// TIA Portal V17 export
// export: Created 2025-06-20T10:18:27.2090798Z, ExportSetting WithDefaults, DisplayName Totally Integrated Automation Portal, DisplayVersion V17 Update 8, DisplayName TIA Portal Openness, DisplayVersion V17 Update 8, DisplayName TIA Portal Version Control Interface, DisplayVersion V17, DisplayName SINAMICS Startdrive Advanced, DisplayVersion V17 SP2, DisplayName SINAMICS Startdrive G110M, G120, G120C, G120D, G120P, G115D, DisplayVersion V17 SP2, DisplayName SINAMICS Startdrive G130, G150, S120, S150, SINAMICS MV, S210, DisplayVersion V17 SP2, DisplayName STEP 7 Professional, DisplayVersion V17 Update 8, DisplayName SINUMERIK ONE STEP 7 Toolbox, DisplayVersion V17 Update 12, DisplayName SINUMERIK ONE PLC Basic Program Plus, DisplayVersion V17 Update 12, DisplayName SINUMERIK 840D sl STEP 7 Toolbox, DisplayVersion V17 Update 12, DisplayName STEP 7 Safety, DisplayVersion V17 Update 6, DisplayName WinCC Advanced, DisplayVersion V17 Update 8
DATA_BLOCK "DB17100_MAINTENANCE_OPERATOR_HELP"   // DB17100
{ S7_Optimized_Access := 'TRUE'; DB_Accessible_From_OPC_UA := 'FALSE' }
VERSION : 0.1
// stored: AutoNumber false, DBAccessibleFromOPCUA false, DBAccessibleFromWebserver true, IsOnlyStoredInLoadMemory false, IsRetainMemResEnabled false, IsWriteProtectedInAS false, MemoryReserve 100
   VAR
      OPERATOR_HELP : Array[0..100] of Bool;
   END_VAR
BEGIN
   // OPERATOR_HELP[0] : MAINTENANCE OPERATOR HELP
   // OPERATOR_HELP[1] : POWDER > UNIT 1 > GENERAL -- UNIT 1 ACTION IN TUBE OF SECTION 4
   // OPERATOR_HELP[2] : POWDER > UNIT 1 > GENERAL -- UNIT 1 ACTION IN TUBE OF SECTION 5
   // OPERATOR_HELP[3] : POWDER > UNIT 1 > GENERAL -- UNIT 1 ACTION IN RIGID TUBE OF THE SPLITTER
   // OPERATOR_HELP[4] : POWDER > UNIT 1 > GENERAL -- UNIT 1 NOZZLE MEDICOAT CALIBRATION
   // OPERATOR_HELP[5] : POWDER > UNIT 1 > GENERAL -- UNIT 1 COMBINER MEDICOAT CALIBRATION
   // OPERATOR_HELP[6] : POWDER > UNIT 1 > GENERAL -- OBTAINING OF UNIT 1 POWDER FLOW (GR/MIN)
   // OPERATOR_HELP[7] : POWDER > UNIT 1 > HOPPER 1 -- ACTION IN UNIT 1 HOPPER 1
   // OPERATOR_HELP[8] : POWDER > UNIT 1 > HOPPER 1 -- ACTION IN PINCHVALVE OF UNIT 1 HOPPER 1
   // OPERATOR_HELP[9] : POWDER > UNIT 1 > HOPPER 1 -- ACTION IN TUBE SECTION 1 OF UNIT 1 HOPPER 1
   // OPERATOR_HELP[10] : POWDER > UNIT 1 > HOPPER 1 -- ACTION IN TUBE SECTION 2 OF UNIT 1 HOPPER 1
   // OPERATOR_HELP[11] : POWDER > UNIT 1 > HOPPER 1 -- UNIT 1 HOPPER 1 LOAD CELL TARE
   // OPERATOR_HELP[12] : POWDER > UNIT 1 > HOPPER 2 -- ACTION IN UNIT 1 HOPPER 2
   // OPERATOR_HELP[13] : POWDER > UNIT 1 > HOPPER 2 -- ACTION IN PINCHVALVE OF UNIT 1 HOPPER 2
   // OPERATOR_HELP[14] : POWDER > UNIT 1 > HOPPER 2 -- ACTION IN TUBE SECTION 1 OF UNIT 1 HOPPER 2
   // OPERATOR_HELP[15] : POWDER > UNIT 1 > HOPPER 2 -- ACTION IN TUBE SECTION 2 OF UNIT 1 HOPPER 2
   // OPERATOR_HELP[16] : POWDER > UNIT 1 > HOPPER 2 -- UNIT 1 HOPPER 2 LOAD CELL TARE
   // OPERATOR_HELP[17] : POWDER > UNIT 1 > FEEDER 1 -- CHANGE OF FEEDER 1 UNIT 1
   // OPERATOR_HELP[18] : POWDER > UNIT 1 > FEEDER 1 -- ACTION IN HOPPER UNIT 1 FEEDER 1 LINE 1
   // OPERATOR_HELP[19] : POWDER > UNIT 1 > FEEDER 1 -- ACTION IN TUBE SECTION 3 UNIT 1 FEEDER 1 LINE 1
   // OPERATOR_HELP[20] : POWDER > UNIT 1 > FEEDER 1 -- ACTION IN HOPPER UNIT 1 FEEDER 1 LINE 2
   // OPERATOR_HELP[21] : POWDER > UNIT 1 > FEEDER 1 -- ACTION IN TUBE SECTION 3 UNIT 1 FEEDER 1 LINE 2
   // OPERATOR_HELP[22] : POWDER > UNIT 1 > FEEDER 1 -- UNIT 1 FEEDER 1 HOPPER 1 TIGHTNESS TEST
   // OPERATOR_HELP[23] : POWDER > UNIT 1 > FEEDER 1 -- UNIT 1 FEEDER 1 HOPPER 2 TIGHTNESS TEST
   // OPERATOR_HELP[24] : POWDER > UNIT 1 > FEEDER 1 -- UNIT 1 LINE 1 MEDICOAT CALIBRATION
   // OPERATOR_HELP[25] : POWDER > UNIT 1 > FEEDER 1 -- UNIT 1 LINE 2 MEDICOAT CALIBRATION
   // OPERATOR_HELP[26] : POWDER > UNIT 2 > GENERAL -- UNIT 2 ACTION IN TUBE OF SECTION 4
   // OPERATOR_HELP[27] : POWDER > UNIT 2 > GENERAL -- UNIT 2 ACTION IN TUBE OF SECTION 5
   // OPERATOR_HELP[28] : POWDER > UNIT 2 > GENERAL -- UNIT 2 ACTION IN RIGID TUBE OF THE SPLITTER
   // OPERATOR_HELP[29] : POWDER > UNIT 2 > GENERAL -- UNIT 2 COMBINER MEDICOAT CALIBRATION
   // OPERATOR_HELP[30] : POWDER > UNIT 2 > GENERAL -- UNIT 2 NOZZLE MEDICOAT CALIBRATION
   // OPERATOR_HELP[31] : POWDER > UNIT 2 > GENERAL -- OBTAINING OF UNIT 2 POWDER FLOW (GR/MIN)
   // OPERATOR_HELP[32] : POWDER > UNIT 2 > HOPPER 1 -- ACTION IN UNIT 2 HOPPER 1
   // OPERATOR_HELP[33] : POWDER > UNIT 2 > HOPPER 1 -- ACTION IN PINCHVALVE OF UNIT 2 HOPPER 1
   // OPERATOR_HELP[34] : POWDER > UNIT 2 > HOPPER 1 -- ACTION IN TUBE SECTION 1 OF UNIT 2 HOPPER 1
   // OPERATOR_HELP[35] : POWDER > UNIT 2 > HOPPER 1 -- ACTION IN TUBE SECTION 2 OF UNIT 2 HOPPER 1
   // OPERATOR_HELP[36] : POWDER > UNIT 2 > HOPPER 1 -- UNIT 2 HOPPER 1 LOAD CELL TARE
   // OPERATOR_HELP[37] : POWDER > UNIT 2 > HOPPER 2 -- ACTION IN UNIT 2 HOPPER 2
   // OPERATOR_HELP[38] : POWDER > UNIT 2 > HOPPER 2 -- ACTION IN PINCHVALVE OF UNIT 2 HOPPER 2
   // OPERATOR_HELP[39] : POWDER > UNIT 2 > HOPPER 2 -- ACTION IN TUBE SECTION 1 OF UNIT 2 HOPPER 2
   // OPERATOR_HELP[40] : POWDER > UNIT 2 > HOPPER 2 -- ACTION IN TUBE SECTION 2 OF UNIT 2 HOPPER 2
   // OPERATOR_HELP[41] : POWDER > UNIT 2 > HOPPER 2 -- UNIT 2 HOPPER 2 LOAD CELL TARE
   // OPERATOR_HELP[42] : POWDER > UNIT 2 > HOPPER 3 -- ACTION IN UNIT 2 HOPPER 3
   // OPERATOR_HELP[43] : POWDER > UNIT 2 > HOPPER 3 -- ACTION IN PINCHVALVE OF UNIT 2 HOPPER 3
   // OPERATOR_HELP[44] : POWDER > UNIT 2 > HOPPER 3 -- ACTION IN TUBE SECTION 1 OF UNIT 2 HOPPER 3
   // OPERATOR_HELP[45] : POWDER > UNIT 2 > HOPPER 3 -- ACTION IN TUBE SECTION 2 OF UNIT 2 HOPPER 3
   // OPERATOR_HELP[46] : POWDER > UNIT 2 > HOPPER 3 -- UNIT 2 HOPPER 3 LOAD CELL TARE
   // OPERATOR_HELP[47] : POWDER > UNIT 2 > FEEDER 1 -- ACTION IN HOPPER UNIT 2 FEEDER 1 LINE 1
   // OPERATOR_HELP[48] : POWDER > UNIT 2 > FEEDER 1 -- ACTION IN TUBE SECTION 3 UNIT 2 FEEDER 1 LINE 1
   // OPERATOR_HELP[49] : POWDER > UNIT 2 > FEEDER 1 -- ACTION IN HOPPER UNIT 2 FEEDER 1 LINE 2
   // OPERATOR_HELP[50] : POWDER > UNIT 2 > FEEDER 1 -- ACTION IN TUBE SECTION 3 UNIT 2 FEEDER 1 LINE 2
   // OPERATOR_HELP[51] : POWDER > UNIT 2 > FEEDER 1 -- UNIT 2 FEEDER 1 HOPPER 1 TIGHTNESS TEST
   // OPERATOR_HELP[52] : POWDER > UNIT 2 > FEEDER 1 -- UNIT 2 FEEDER 1 HOPPER 2 TIGHTNESS TEST
   // OPERATOR_HELP[53] : POWDER > UNIT 2 > FEEDER 1 -- UNIT 2 LINE 1 MEDICOAT CALIBRATION
   // OPERATOR_HELP[54] : POWDER > UNIT 2 > FEEDER 1 -- UNIT 2 LINE 2 MEDICOAT CALIBRATION
   // OPERATOR_HELP[55] : POWDER > UNIT 2 > FEEDER 2 -- ACTION IN HOPPER UNIT 2 FEEDER 2 LINE 3
   // OPERATOR_HELP[56] : POWDER > UNIT 2 > FEEDER 2 -- ACTION IN TUBE SECTION 3 UNIT 2 FEEDER 2 LINE 3
   // OPERATOR_HELP[57] : POWDER > UNIT 2 > FEEDER 2 -- UNIT 2 FEEDER 2 HOPPER 2 TIGHTNESS TEST
   // OPERATOR_HELP[58] : POWDER > UNIT 2 > FEEDER 2 -- UNIT 2 LINE 2 MEDICOAT CALIBRATION
   // OPERATOR_HELP[59] : MACHINE > UNIT 1 > GENERAL -- CHECK UNIT 1 FIXTURE 1
   // OPERATOR_HELP[60] : MACHINE > UNIT 1 > GENERAL -- CHECK UNIT 1 FIXTURE 2
   // OPERATOR_HELP[61] : MACHINE > UNIT 1 > GENERAL -- CHECK UNIT 1 FIXTURE 3
   // OPERATOR_HELP[62] : MACHINE > UNIT 1 > GENERAL -- CHECK UNIT 1 FIXTURE 4
   // OPERATOR_HELP[63] : MACHINE > UNIT 1 > GENERAL -- CHANGE IN UNIT 1 STATION 3 SEALING SYSTEM
   // OPERATOR_HELP[64] : MACHINE > UNIT 1 > GENERAL -- ADJUST UNIT 1 LASER HEAD (RADIAL / TANGENTIAL ANGLES)
   // OPERATOR_HELP[65] : MACHINE > UNIT 1 > GENERAL -- UNIT 1 STATION 3 PROFILOMETER CALIBRATION
   // OPERATOR_HELP[66] : MACHINE > UNIT 1 > GENERAL -- UNIT 1 CAMERA ADJUSTMENT SEQUENCE
   // OPERATOR_HELP[67] : MACHINE > UNIT 1 > GENERAL -- UNIT 1 CLEANING PERFILOMETER LENT
   // OPERATOR_HELP[68] : MACHINE > UNIT 1 > GENERAL -- UNIT 1 CONFIGURATION OF PYROMETER ON GOING
   // OPERATOR_HELP[69] : MACHINE > UNIT 1 > GENERAL -- UNIT 1 CHANGE IN WATER SYSTEM
   // OPERATOR_HELP[70] : MACHINE > UNIT 1 > GENERAL -- UNIT 1 CHANGE IN GAS SYSTEM
   // OPERATOR_HELP[71] : MACHINE > UNIT 1 > GENERAL -- UNIT 1 AXIS REFERENCE SEQUENCE
   // OPERATOR_HELP[72] : MACHINE > UNIT 1 > GENERAL -- UNIT 1 AXIS C11 CHANGE
   // OPERATOR_HELP[73] : MACHINE > UNIT 1 > GENERAL -- UNIT 1 AXIS C12 CHANGE
   // OPERATOR_HELP[74] : MACHINE > UNIT 1 > GENERAL -- UNIT 1 AXIS C13 CHANGE
   // OPERATOR_HELP[75] : MACHINE > UNIT 1 > GENERAL -- UNIT 1 AXIS C14 CHANGE
   // OPERATOR_HELP[76] : MACHINE > UNIT 1 > GENERAL -- UNIT 1 AXIS X13 CHANGE
   // OPERATOR_HELP[77] : MACHINE > UNIT 1 > GENERAL -- UNIT 1 AXIS Z13 CHANGE
   // OPERATOR_HELP[78] : MACHINE > UNIT 1 > GENERAL -- UNIT 1 AXIS E10 CHANGE
   // OPERATOR_HELP[79] : MACHINE > UNIT 1 > LASER -- CHECK UNIT 1 NOZZLE
   // OPERATOR_HELP[80] : MACHINE > UNIT 2 > GENERAL -- CHECK UNIT 2 FIXTURE 1
   // OPERATOR_HELP[81] : MACHINE > UNIT 2 > GENERAL -- CHECK UNIT 2 FIXTURE 2
   // OPERATOR_HELP[82] : MACHINE > UNIT 2 > GENERAL -- CHECK UNIT 2 FIXTURE 3
   // OPERATOR_HELP[83] : MACHINE > UNIT 2 > GENERAL -- CHECK UNIT 2 FIXTURE 4
   // OPERATOR_HELP[84] : MACHINE > UNIT 2 > GENERAL -- CHANGE IN UNIT 2 STATION 3 SEALING SYSTEM
   // OPERATOR_HELP[85] : MACHINE > UNIT 2 > GENERAL -- ADJUST UNIT 2 LASER HEAD (RADIAL / TANGENTIAL ANGLES)
   // OPERATOR_HELP[86] : MACHINE > UNIT 2 > GENERAL -- UNIT 2 STATION 3 PROFILOMETER CALIBRATION
   // OPERATOR_HELP[87] : MACHINE > UNIT 2 > GENERAL -- UNIT 2 CAMERA ADJUSTMENT SEQUENCE
   // OPERATOR_HELP[88] : MACHINE > UNIT 2 > GENERAL -- UNIT 2 CLEANING PERFILOMETER LENT
   // OPERATOR_HELP[89] : MACHINE > UNIT 2 > GENERAL -- UNIT 2 CONFIGURATION OF PYROMETER ON GOING
   // OPERATOR_HELP[90] : MACHINE > UNIT 2 > GENERAL -- UNIT 2 CHANGE IN WATER SYSTEM
   // OPERATOR_HELP[91] : MACHINE > UNIT 2 > GENERAL -- UNIT 2 CHANGE IN GAS SYSTEM
   // OPERATOR_HELP[92] : MACHINE > UNIT 2 > GENERAL -- UNIT 2 AXIS REFERENCE SEQUENCE
   // OPERATOR_HELP[93] : MACHINE > UNIT 2 > GENERAL -- UNIT 2 AXIS C21 CHANGE
   // OPERATOR_HELP[94] : MACHINE > UNIT 2 > GENERAL -- UNIT 2 AXIS C22 CHANGE
   // OPERATOR_HELP[95] : MACHINE > UNIT 2 > GENERAL -- UNIT 2 AXIS C23 CHANGE
   // OPERATOR_HELP[96] : MACHINE > UNIT 2 > GENERAL -- UNIT 2 AXIS C24 CHANGE
   // OPERATOR_HELP[97] : MACHINE > UNIT 2 > GENERAL -- UNIT 2 AXIS X23 CHANGE
   // OPERATOR_HELP[98] : MACHINE > UNIT 2 > GENERAL -- UNIT 2 AXIS Z23 CHANGE
   // OPERATOR_HELP[99] : MACHINE > UNIT 2 > GENERAL -- UNIT 2 AXIS E20 CHANGE
   // OPERATOR_HELP[100] : MACHINE > UNIT 2 > LASER -- CHECK UNIT 2 NOZZLE
END_DATA_BLOCK
